// TIA Portal V19 export
DATA_BLOCK "PPrgArchive20"   // DB517
// stored: IsOnlyStoredInLoadMemory true, MemoryReserve 0, Namespace G
   VAR RETAIN
      PRG : Array[1901..2000] of "PPrg_Data";
   END_VAR
BEGIN
END_DATA_BLOCK
